TYPE CM_Sensor_STS :
STRUCT
	Tag				: STRING;
	Output			: BOOL;
	Auto			: BOOL;
	Manueel			: BOOL;
END_STRUCT
END_TYPE

(* stored: Version 1.1.0.1, ProductVersion 3.1.4024.12
   DUT CM_Sensor_STS: Id {a3a52ed6-76eb-4eda-86b6-3df088bed856} *)
